(* PLC project trigger_function, Dassault Systèmes ControlBuild 2024x *)
(* stored: creationDateTime 2023-10-04T11:03:52-01:00 *)

FUNCTION_BLOCK motion_lib.trigger_function
  VAR_INPUT
    armExtrem : ARRAY[1..3] OF REAL := [3(0.0)];
    productId : DINT := -1;
  END_VAR
  VAR_OUTPUT
    velX : REAL := 0.0;
    velY : REAL := 0.0;
    velZ : REAL := 0.0;
    armInStop : BOOL := false;
  END_VAR
  VAR
    armExtrem1 : ARRAY[1..3] OF REAL := [3(0.0)];
    i : INT := 0;
    productTimeDetect : REAL := 0.0;
    productDetected : BOOL := false;
    productId1 : DINT := -1;
    actionTake : BOOL := false;
    activeArea : BOOL := false;
  END_VAR
  VAR CONSTANT
    ACTIVE_AREA_Z : REAL := 1100.0;
    TEMPO_DETECTION_PRO : REAL := 0.2;
  END_VAR


ACTION C_source_code:
if (productId1 == -1 && productId != -1) 
	productTimeDetect = 0;

if (productId != -1) 
	productTimeDetect += CLOCK_PERIOD / 1000000;

if (productTimeDetect > TEMPO_DETECTION_PRO) productDetected = 1; else productDetected = 0;

velX = 1000000 * (armExtrem(1) - armExtrem1(1)) / CLOCK_PERIOD; // mm/s
velY = 1000000 * (armExtrem(2) - armExtrem1(2)) / CLOCK_PERIOD;
velZ = 1000000 * (armExtrem(3) - armExtrem1(3)) / CLOCK_PERIOD;

armInStop = (fabs(velX) < 10 && fabs(velY) < 10 && velZ < -50);



for (i = 1; i <= 3; i++)
	armExtrem1(i) = armExtrem(i);

productId1 = productId;
END_ACTION
END_FUNCTION_BLOCK
